ABB RobotStudio station: solution.rsstn

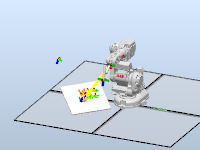
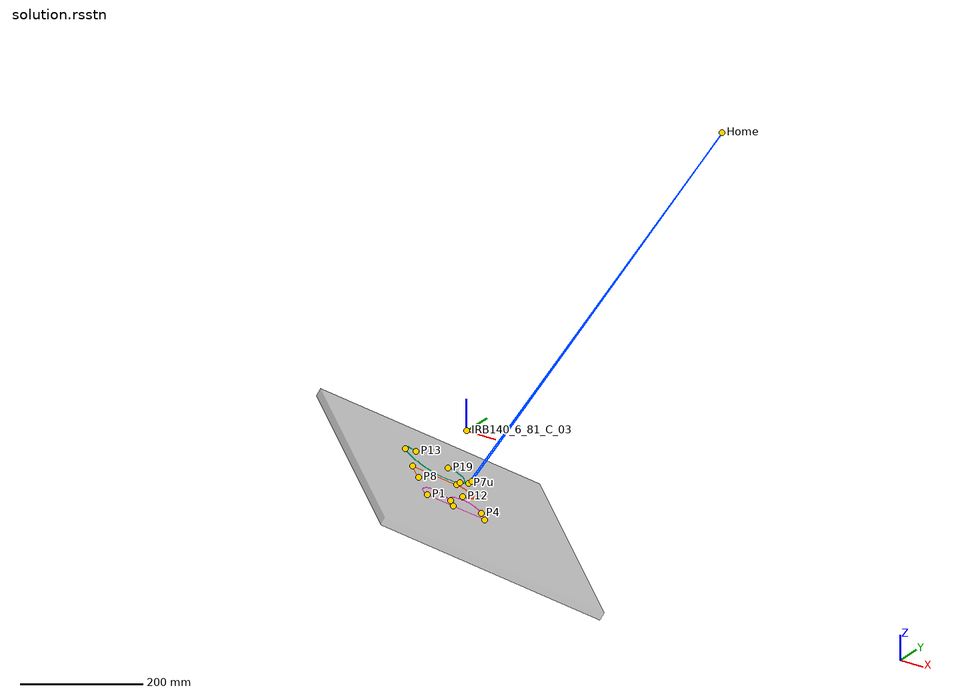
[picture v1: parts stored in the station drawn from their meshes, with robot base, taught points and paths (robot models come from the ABB library and are not in the file)]
Station solution (saved by RobotStudio 22.1.9826.0)
Controller ControllerIRC5
  mechanical unit ROB_1: IRB140_6_81_C_03, 6 joints, base frame (0, 0, 0) mm
Layout (positions relative to the parent item):
  - IRB140_6_81_C_03 [mechanism, from Robots\IRB140_6_81_C_G_03.rslib] at (0, 0, 0) mm; joint values [0, 0, 0, -3.1416, -0.5236, 3.1416] (rad or m)
  - MarkerPenTool [mechanism, from lib\MarkerPenTool.rslib] at (506.29, 0, 679.5) mm, rotated rx 180 ry 60 rz 180 deg
  - Base [part] at (583.92, -444.71, 12.17) mm, rotated rx -60 ry 0 rz 137.35 deg, size 490 x 14 x 420 mm
Attachment: MarkerPenTool is attached to IRB140_6_81_C_03 / Link6
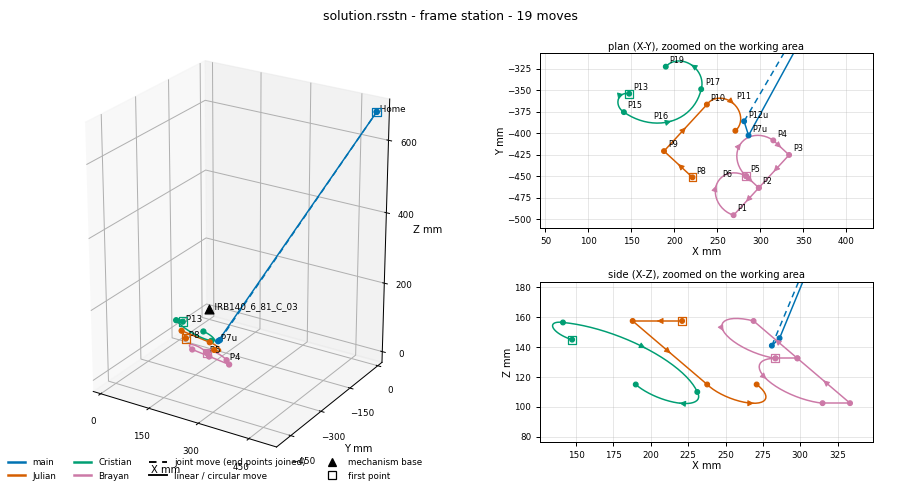
[picture p0: tool path of solution.rsstn in frame station, 19 of 19 moves have a stored position in this frame; points joined in program order, loops and branches not executed]
Targets, tools, work objects and paths stored in the station, written as RAPID:
! task T_ROB1
MODULE CalibData
  PERS tooldata MarkerPenTool:=[TRUE,[[12.566,0,214.048],[0.000228956,0.382764099,0.000092128,0.923846082]],[0.162,[-27,0,110],[1,0,0,0],0.003,0.003,0.0003162]];
  PERS tooldata toolBJC:=[TRUE,[[12.254,-0.002,214.736],[0.923879533,0,0.382683432,0]],[0.162,[-27.13,0,109.8621],[1,0,0,0],0.003,0.003,0.0003162]];
  TASK PERS wobjdata whiteBoard:=[FALSE,TRUE,"",[[373.72422246,-432.807039289,90.000000038],[0.351258535,0.094119441,0.24109921,0.899794501]],[[0,0,0],[1,0,0,0]]];
ENDMODULE

! task T_ROB1
MODULE BJC
  CONST robtarget Home:=[[506.292,0,679.5],[0.5,0,0.866025404,0],[0,-1,0,1],[9E+09,9E+09,9E+09,9E+09,9E+09,9E+09]];
  CONST robtarget P7u:=[[85,60,30],[0,0.707106781,0.707106781,0],[0,-1,0,1],[9E+09,9E+09,9E+09,9E+09,9E+09,9E+09]];
  CONST robtarget P12u:=[[100,50,30],[0,0.707106781,0.707106781,0],[0,-1,0,1],[9E+09,9E+09,9E+09,9E+09,9E+09,9E+09]];
  CONST robtarget P8:=[[100,135,0],[0,0.707106781,0.707106781,0],[0,-1,0,1],[9E+09,9E+09,9E+09,9E+09,9E+09,9E+09]];
  CONST robtarget P9:=[[145,135,0],[0,0.707106781,0.707106781,0],[0,-1,0,1],[9E+09,9E+09,9E+09,9E+09,9E+09,9E+09]];
  CONST robtarget P10:=[[145,50,0],[0,0.707106781,0.707106781,0],[0,-1,0,1],[9E+09,9E+09,9E+09,9E+09,9E+09,9E+09]];
  CONST robtarget P11:=[[125,25,0],[0,0.707106781,0.707106781,0],[0,-1,0,1],[9E+09,9E+09,9E+09,9E+09,9E+09,9E+09]];
  CONST robtarget P12:=[[100,50,0],[0,0.707106781,0.707106781,0],[0,-1,0,1],[9E+09,9E+09,9E+09,9E+09,9E+09,9E+09]];
  CONST robtarget P13:=[[220,110,0],[0,0.707106781,0.707106781,0],[0,-1,0,1],[9E+09,9E+09,9E+09,9E+09,9E+09,9E+09]];
  CONST robtarget P14:=[[225,125,0],[0,0.707106781,0.707106781,0],[0,-1,0,1],[9E+09,9E+09,9E+09,9E+09,9E+09,9E+09]];
  CONST robtarget P15:=[[210,133,0],[0,0.707106781,0.707106781,0],[0,-1,0,1],[9E+09,9E+09,9E+09,9E+09,9E+09,9E+09]];
  CONST robtarget P16:=[[180,120,0],[0,0.707106781,0.707106781,0],[0,-1,0,1],[9E+09,9E+09,9E+09,9E+09,9E+09,9E+09]];
  CONST robtarget P17:=[[162,40,0],[0,0.707106781,0.707106781,0],[0,-1,0,1],[9E+09,9E+09,9E+09,9E+09,9E+09,9E+09]];
  CONST robtarget P18:=[[190,25,0],[0,0.707106781,0.707106781,0],[0,-1,0,1],[9E+09,9E+09,9E+09,9E+09,9E+09,9E+09]];
  CONST robtarget P19:=[[210,50,0],[0,0.707106781,0.707106781,0],[0,-1,0,1],[9E+09,9E+09,9E+09,9E+09,9E+09,9E+09]];
  CONST robtarget P5:=[[55,85,0],[0,0.707106781,0.707106781,0],[0,-1,0,1],[9E+09,9E+09,9E+09,9E+09,9E+09,9E+09]];
  CONST robtarget P2:=[[35,85,0],[0,0.707106781,0.707106781,0],[0,-1,0,1],[9E+09,9E+09,9E+09,9E+09,9E+09,9E+09]];
  CONST robtarget P1:=[[35,135,0],[0,0.707106781,0.707106781,0],[0,-1,0,1],[9E+09,9E+09,9E+09,9E+09,9E+09,9E+09]];
  CONST robtarget P6:=[[75,115,0],[0,0.707106781,0.707106781,0],[0,-1,0,1],[9E+09,9E+09,9E+09,9E+09,9E+09,9E+09]];
  CONST robtarget P7:=[[85,60,0],[0,0.707106781,0.707106781,0],[0,-1,0,1],[9E+09,9E+09,9E+09,9E+09,9E+09,9E+09]];
  CONST robtarget P4:=[[60,25,0],[0,0.707106781,0.707106781,0],[0,-1,0,1],[9E+09,9E+09,9E+09,9E+09,9E+09,9E+09]];
  CONST robtarget P3:=[[35,25,0],[0,0.707106781,0.707106781,0],[0,-1,0,1],[9E+09,9E+09,9E+09,9E+09,9E+09,9E+09]];
  PROC main()
    MoveJ Home,v1000,z100,tool0;
    Brayan;
    MoveL P7u,v1000,z0,toolBJC\WObj:=whiteBoard;
    Julian;
    MoveL P12u,v1000,z0,toolBJC\WObj:=whiteBoard;
    Cristian;
    MoveJ Home,v1000,z0,tool0;
  ENDPROC
  PROC Julian()
    MoveJ P8,v1000,z0,toolBJC\WObj:=whiteBoard;
    MoveL P9,v100,z0,toolBJC\WObj:=whiteBoard;
    MoveL P10,v100,z0,toolBJC\WObj:=whiteBoard;
    MoveC P11,P12,v100,z0,toolBJC\WObj:=whiteBoard;
  ENDPROC
  PROC Cristian()
    MoveJ P13,v1000,z0,toolBJC\WObj:=whiteBoard;
    MoveC P14,P15,v100,z0,toolBJC\WObj:=whiteBoard;
    MoveC P16,P17,v100,z0,toolBJC\WObj:=whiteBoard;
    MoveC P18,P19,v100,z0,toolBJC\WObj:=whiteBoard;
  ENDPROC
  PROC Brayan()
    MoveJ P5,v1000,z0,toolBJC\WObj:=whiteBoard;
    MoveL P2,v100,z0,toolBJC\WObj:=whiteBoard;
    MoveL P1,v100,z0,toolBJC\WObj:=whiteBoard;
    MoveC P6,P5,v100,z0,toolBJC\WObj:=whiteBoard;
    MoveC P7,P4,v100,z0,toolBJC\WObj:=whiteBoard;
    MoveL P3,v100,z0,toolBJC\WObj:=whiteBoard;
    MoveL P2,v100,z0,toolBJC\WObj:=whiteBoard;
  ENDPROC
ENDMODULE

! task T_ROB1
MODULE Module1
  CONST robtarget Target_10:=[[-294.402671987,271.820134726,536.519754089],[0.04746601,0.923566415,0.360538473,-0.121589741],[-1,-2,2,1],[9E+09,9E+09,9E+09,9E+09,9E+09,9E+09]];
  CONST robtarget Target_20:=[[-294.402671987,271.820134726,536.519754089],[0.04746601,0.923566415,0.360538473,-0.121589741],[-1,-2,2,1],[9E+09,9E+09,9E+09,9E+09,9E+09,9E+09]];
ENDMODULE

